PROGRAM Safety_Template
VAR
END_VAR

//Define parameters of safety device
(*IF _TaskInfo[fbGetCurTaskIndex.index].FirstCycle THEN
	astSafety[1].stSafetyDescription.sSafetyName := 'Light Curtain 1';
	astSafety[1].stSafetyDescription.sLocation := 'Up stream';
	astSafety[1].stSafetyDescription.eSafetyType := E_SafetyType.eSingleChannel;
END_IF*)

END_PROGRAM

(* stored: Version 1.1.0.1, ProductVersion 3.1.4024.11
   POU Safety_Template: Id {3c734c42-54fb-4db2-a966-7fb15fcc6c35}, SpecialFunc None *)
